// TIA Portal V19 export
ORGANIZATION_BLOCK "Main_Switch"   // OB123, LAD, ProgramCycle
TITLE = "Main Program Sweep (Cycle)"
{ S7_Optimized_Access := 'TRUE' }
// stored: AutoNumber false, SetENOAutomatically false
   VAR_INPUT
      Initial_Call : Bool;   // Initial call of this OB
      Remanence : Bool;   // =True, if remanent data are available
   END_VAR
   VAR_TEMP
      retvalue : Int;
      text : String;
      retVal : Word;
      Busy : Bool;
   END_VAR
   VAR_TEMP   // added for the SCL form of the ladder/FBD networks
      _w1 : Bool;
   END_VAR
BEGIN

REGION Network 1: Cycle Measurement - Tic
   // Scan and store but only to reset the runtime counter at the top of the scan. the Ret_Val is collected at the end of the program cycle or area of focus.
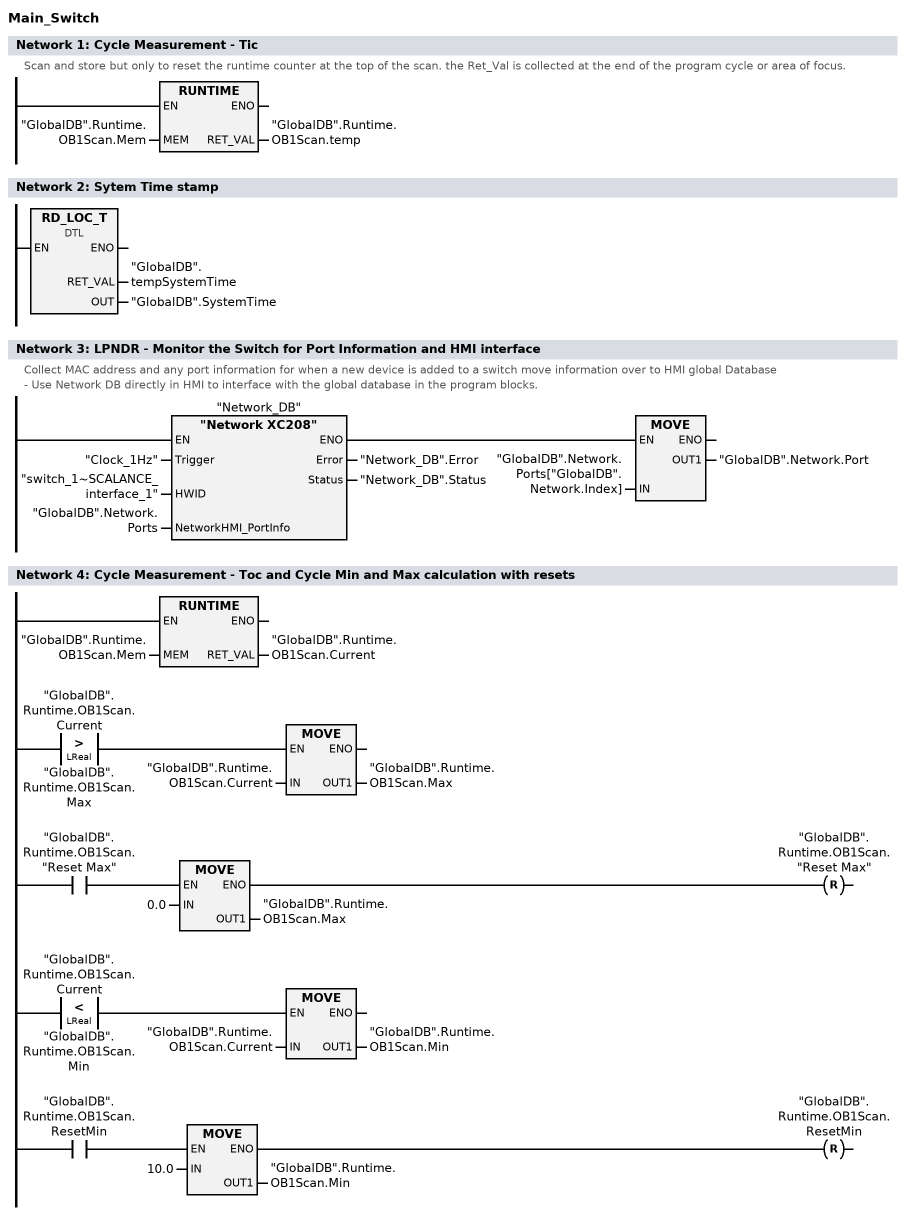
   // no SCL statement known for Runtime: written as a call
   "GlobalDB".Runtime.OB1Scan.temp := Runtime(mem := "GlobalDB".Runtime.OB1Scan.Mem);
END_REGION

REGION Network 2: Sytem Time stamp
   RUNG wire#powerrail
      { S7_Templates := "date_type := DTL" } RD_LOC_T(RET_VAL => "GlobalDB".tempSystemTime, OUT => "GlobalDB".SystemTime)
   END_RUNG
   // the same network as SCL:
   "GlobalDB".tempSystemTime := RD_LOC_T(OUT => "GlobalDB".SystemTime);
END_REGION

REGION Network 3: LPNDR - Monitor the Switch for Port Information and HMI interface
   // Collect MAC address and any port information for when a new device is added to a switch move information over to HMI global Database
   // 
   // - Use Network DB directly in HMI to interface with the global database in the program blocks.
   RUNG wire#powerrail
      "Network_DB"(Trigger := "Clock_1Hz", HWID := "switch_1~SCALANCE_interface_1", NetworkHMI_PortInfo := "GlobalDB".Network.Ports, Error => "Network_DB".Error, Status => "Network_DB".Status)
      Move(in := "GlobalDB".Network.Ports["GlobalDB".Network.Index], out1 => "GlobalDB".Network.Port)
   END_RUNG
   // the same network as SCL:
   "Network_DB"(Trigger := "Clock_1Hz",   // "Network XC208"
                HWID := "switch_1~SCALANCE_interface_1",
                NetworkHMI_PortInfo := "GlobalDB".Network.Ports,
                Error => "Network_DB".Error,
                Status => "Network_DB".Status,
                ENO => #_w1);
   IF #_w1 THEN "GlobalDB".Network.Port := "GlobalDB".Network.Ports["GlobalDB".Network.Index]; END_IF;
END_REGION

REGION Network 4: Cycle Measurement - Toc and Cycle Min and Max calculation with resets
   // no SCL statement known for Runtime: written as a call
   "GlobalDB".Runtime.OB1Scan.Current := Runtime(mem := "GlobalDB".Runtime.OB1Scan.Mem);
   IF "GlobalDB".Runtime.OB1Scan.Current > "GlobalDB".Runtime.OB1Scan.Max THEN
       "GlobalDB".Runtime.OB1Scan.Max := "GlobalDB".Runtime.OB1Scan.Current;
   END_IF;
   IF "GlobalDB".Runtime.OB1Scan."Reset Max" THEN
       "GlobalDB".Runtime.OB1Scan.Max := 0.0;
       "GlobalDB".Runtime.OB1Scan."Reset Max" := FALSE;
   END_IF;
   IF "GlobalDB".Runtime.OB1Scan.Current < "GlobalDB".Runtime.OB1Scan.Min THEN
       "GlobalDB".Runtime.OB1Scan.Min := "GlobalDB".Runtime.OB1Scan.Current;
   END_IF;
   IF "GlobalDB".Runtime.OB1Scan.ResetMin THEN
       "GlobalDB".Runtime.OB1Scan.Min := 10.0;
       "GlobalDB".Runtime.OB1Scan.ResetMin := FALSE;
   END_IF;
END_REGION
END_ORGANIZATION_BLOCK
